{attribute 'qualified_only'}
{attribute 'strict'}
TYPE E_EventSorting :
(
	Ascending,		// Oldest to newest Event
	Descending		// Newest to oldest Event
);
END_TYPE

(* stored: Version 1.1.0.1, ProductVersion 3.1.4024.12
   EnumerationTextList E_EventSorting: Id {2545c156-2796-40f9-975f-b90f9744faad} *)
